FUNCTION_BLOCK FB_ReactorSet
VAR_INPUT
	i_seq_req 				: E_RS_SeqState;
	i_cooling_pump_sts 		: ST_Util_Service_Sts;
	i_deadair_pump_sts 		: ST_Util_Service_Sts;
	i_steam_system_sts 		: ST_Util_Service_Sts;
	i_purge_assist_sts		: ST_Util_Service_Sts;	
	i_cooling_pump_assigned : BOOL;
	i_deadair_pump_assigned	: BOOL;
	i_steam_system_assigned	: BOOL;
	i_purge_assist_assigned	: BOOL;
	i_reset_fault			: BOOL;
	
END_VAR
VAR_OUTPUT
	o_adsorption_seq_sts 	: ST_SeqSts;
	o_evac_seq_sts 			: ST_SeqSts;
	o_desorption_seq_sts 	: ST_SeqSts;
	o_cooling_seq_sts 		: ST_SeqSts;
	o_airpress_seq_sts 		: ST_SeqSts;
	
	o_cooling_pump_req		: BYTE;  
	o_deadair_pump_req		: BYTE;
	o_steam_system_req		: BYTE;
	o_purge_assist_req		: BYTE;
	
	o_error_active			: BOOL;
END_VAR
VAR
	
	// from RS Controller 
	in_adsorption_seq_sts  	AT %I*	: BYTE;
	in_evac_seq_sts 		AT %I*	: BYTE;
	in_desorption_seq_sts 	AT %I*	: BYTE;
	in_cooling_seq_sts 		AT %I*	: BYTE;
	in_airpress_seq_sts 	AT %I*	: BYTE;
	
	in_cooling_pump_req		AT %I*	: BYTE;  
	in_deadair_pump_req		AT %I*	: BYTE;
	in_steam_system_req		AT %I*	: BYTE;
	in_purge_assist_req		AT %I*	: BYTE;
	
	in_error_sts			AT %I* 	: BOOL;
	in_error_code1			AT %I*	: DWORD;
	in_error_code2			AT %I*	: DWORD;
	
	
	// to RS Controller
	out_seq_req 				AT %Q*	: BYTE;
	
	out_cooling_pump_sts 		AT %Q*	: BYTE;  
	out_deadair_pump_sts		AT %Q*	: BYTE;
	out_steam_system_sts		AT %Q*	: BYTE;
	out_purge_assist_sts		AT %Q*	: BYTE;
	
	out_cooling_pump_assigned 		AT %Q* : BOOL;
	out_deadair_pump_assigned		AT %Q*: BOOL;
	out_steam_system_assigned		AT %Q*: BOOL;
	out_purge_assist_assigned		AT %Q*: BOOL;
	
	out_error_reset				AT %Q* : BOOL;
	
	
	
	
END_VAR

// Sequence Select + Run request to RS controller

out_seq_req := TO_BYTE(i_seq_req);

// Service Request Assigned Sts to RS Controller

out_cooling_pump_assigned	:= i_cooling_pump_assigned;
out_deadair_pump_assigned	:= i_deadair_pump_assigned;
out_steam_system_assigned	:= i_steam_system_assigned;
out_purge_assist_assigned	:= i_purge_assist_assigned;

// Utilities Services Status  to RS Copntroller 

Set_Service_Sts ( i_service_sts := i_cooling_pump_sts,o_service_sts => out_cooling_pump_sts);
Set_Service_Sts ( i_service_sts := i_deadair_pump_sts,o_service_sts => out_deadair_pump_sts);
Set_Service_Sts ( i_service_sts := i_steam_system_sts,o_service_sts => out_steam_system_sts);
Set_Service_Sts ( i_service_sts := i_purge_assist_sts,o_service_sts => out_purge_assist_sts);

//

// Seq Status from RS controller 

F_Get_Seq_Status(i_seq_sts := in_adsorption_seq_sts,o_seq_sts => o_adsorption_seq_sts);
F_Get_Seq_Status(i_seq_sts := in_evac_seq_sts,o_seq_sts => o_evac_seq_sts);
F_Get_Seq_Status(i_seq_sts := in_desorption_seq_sts,o_seq_sts => o_desorption_seq_sts);
F_Get_Seq_Status(i_seq_sts := in_cooling_seq_sts,o_seq_sts => o_cooling_seq_sts);
F_Get_Seq_Status(i_seq_sts := in_airpress_seq_sts,o_seq_sts => o_airpress_seq_sts);

// Utilities Req from RS Controller 

o_cooling_pump_req		:= in_cooling_pump_req;
o_deadair_pump_req		:= in_deadair_pump_req;
o_steam_system_req		:= in_steam_system_req;
o_purge_assist_req		:= in_purge_assist_req;

// Error mapping from RS Controller
o_error_active := in_error_sts;

// Error reset command to RS Controller
out_error_reset := i_reset_fault;

PROPERTY Reset_Fault : BOOL
SET
out_error_reset := Reset_Fault;
END_SET
END_PROPERTY

METHOD Set_Service_Sts : BOOL
VAR_INPUT
	i_service_sts : ST_Util_Service_Sts;
END_VAR
VAR_OUTPUT
	o_service_sts	: BYTE;
END_VAR
IF i_service_sts.ready THEN
	o_service_sts := 1 ;
ELSIF i_service_sts.running THEN
	o_service_sts := 2 ;
ELSIF i_service_sts.faulted THEN
	o_service_sts := 9 ;
ELSE
	o_service_sts := 0 ;	
END_IF
END_METHOD

END_FUNCTION_BLOCK

(* stored: Version 1.1.0.1, ProductVersion 3.1.4024.12
   POU FB_ReactorSet: Id {8e27e1de-b4c9-47f4-af94-ac0054b8b104}, SpecialFunc None
   Property Reset_Fault: Id {5dc63ca5-d894-4224-9a66-7976dd1ee88e}
   Set Set: Id {2a8619fb-2f3c-44d9-8a80-ad7ac89ad13e}
   Method Set_Service_Sts: Id {7bc84eef-0834-4c67-8959-d790ac013a0b} *)
